{attribute 'GeneratedUsingTerminal: EL3742-0000-0002'}
{attribute addProperty BoxType "EL3742-0000-0002"}
{attribute addProperty Id "EtcSlaveTerminalBaseCh1_CycleCountAT %I*Ch1_CycleCount_9DBE2BC52Ch1_Sample_0AT %I*Ch1_Sample_A71DD5012Ch1_Sample_1AT %I*Ch1_Sample_A71DD5012Ch1_Sample_2AT %I*Ch1_Sample_A71DD5012Ch1_Sample_3AT %I*Ch1_Sample_A71DD5012Ch1_Sample_4AT %I*Ch1_Sample_A71DD5012Ch1_Sample_5AT %I*Ch1_Sample_A71DD5012Ch1_Sample_6AT %I*Ch1_Sample_A71DD5012Ch1_Sample_7AT %I*Ch1_Sample_A71DD5012Ch1_Sample_8AT %I*Ch1_Sample_A71DD5012Ch1_Sample_9AT %I*Ch1_Sample_A71DD5012Ch2_CycleCountAT %I*Ch2_CycleCount_976A51B52Ch2_Sample_0AT %I*Ch2_Sample_9F6886E62Ch2_Sample_1AT %I*Ch2_Sample_9F6886E62Ch2_Sample_2AT %I*Ch2_Sample_9F6886E62Ch2_Sample_3AT %I*Ch2_Sample_9F6886E62Ch2_Sample_4AT %I*Ch2_Sample_9F6886E62Ch2_Sample_5AT %I*Ch2_Sample_9F6886E62Ch2_Sample_6AT %I*Ch2_Sample_9F6886E62Ch2_Sample_7AT %I*Ch2_Sample_9F6886E62Ch2_Sample_8AT %I*Ch2_Sample_9F6886E62Ch2_Sample_9AT %I*Ch2_Sample_9F6886E62WcStateAT %I*WcState_9091E0EB2InfoDataAT %I*InfoData_A7436BC610"}
{attribute addProperty CRC "2340106502"}
{attribute addProperty Size "56"}
TYPE EL3742_8B7B3106 EXTENDS EtcSlaveTerminalBase :
STRUCT
	{attribute addProperty Name "Ch1_CycleCount"}
	Ch1_CycleCount : Ch1_CycleCount_9DBE2BC5;
	{attribute addProperty Name "Ch1_Sample_0"}
	Ch1_Sample_0 : Ch1_Sample_A71DD501;
	{attribute addProperty Name "Ch1_Sample_1"}
	Ch1_Sample_1 : Ch1_Sample_A71DD501;
	{attribute addProperty Name "Ch1_Sample_2"}
	Ch1_Sample_2 : Ch1_Sample_A71DD501;
	{attribute addProperty Name "Ch1_Sample_3"}
	Ch1_Sample_3 : Ch1_Sample_A71DD501;
	{attribute addProperty Name "Ch1_Sample_4"}
	Ch1_Sample_4 : Ch1_Sample_A71DD501;
	{attribute addProperty Name "Ch1_Sample_5"}
	Ch1_Sample_5 : Ch1_Sample_A71DD501;
	{attribute addProperty Name "Ch1_Sample_6"}
	Ch1_Sample_6 : Ch1_Sample_A71DD501;
	{attribute addProperty Name "Ch1_Sample_7"}
	Ch1_Sample_7 : Ch1_Sample_A71DD501;
	{attribute addProperty Name "Ch1_Sample_8"}
	Ch1_Sample_8 : Ch1_Sample_A71DD501;
	{attribute addProperty Name "Ch1_Sample_9"}
	Ch1_Sample_9 : Ch1_Sample_A71DD501;
	{attribute addProperty Name "Ch2_CycleCount"}
	Ch2_CycleCount : Ch2_CycleCount_976A51B5;
	{attribute addProperty Name "Ch2_Sample_0"}
	Ch2_Sample_0 : Ch2_Sample_9F6886E6;
	{attribute addProperty Name "Ch2_Sample_1"}
	Ch2_Sample_1 : Ch2_Sample_9F6886E6;
	{attribute addProperty Name "Ch2_Sample_2"}
	Ch2_Sample_2 : Ch2_Sample_9F6886E6;
	{attribute addProperty Name "Ch2_Sample_3"}
	Ch2_Sample_3 : Ch2_Sample_9F6886E6;
	{attribute addProperty Name "Ch2_Sample_4"}
	Ch2_Sample_4 : Ch2_Sample_9F6886E6;
	{attribute addProperty Name "Ch2_Sample_5"}
	Ch2_Sample_5 : Ch2_Sample_9F6886E6;
	{attribute addProperty Name "Ch2_Sample_6"}
	Ch2_Sample_6 : Ch2_Sample_9F6886E6;
	{attribute addProperty Name "Ch2_Sample_7"}
	Ch2_Sample_7 : Ch2_Sample_9F6886E6;
	{attribute addProperty Name "Ch2_Sample_8"}
	Ch2_Sample_8 : Ch2_Sample_9F6886E6;
	{attribute addProperty Name "Ch2_Sample_9"}
	Ch2_Sample_9 : Ch2_Sample_9F6886E6;
	{attribute addProperty Name "WcState"}
	WcState : WcState_9091E0EB;
	{attribute addProperty Name "InfoData"}
	InfoData : InfoData_A7436BC6;
END_STRUCT
END_TYPE

(* stored: Version 1.2.0.0, ProductVersion 3.1.4024.9
   DUT EL3742_8B7B3106: Id {d3076b7d-7c76-45cf-921e-5c0ee7536fcc} *)
